{attribute 'qualified_only'}
{attribute 'strict'}
TYPE eSavePositionOnPLC :
(
	ePostionHardDisk := 0,
	ePostionC := 1
);
END_TYPE

(* stored: Version 1.1.0.1, ProductVersion 3.1.4024.9
   DUT eSavePositionOnPLC: Id {b0e034bd-8d78-4415-b724-947a67d2504f} *)
